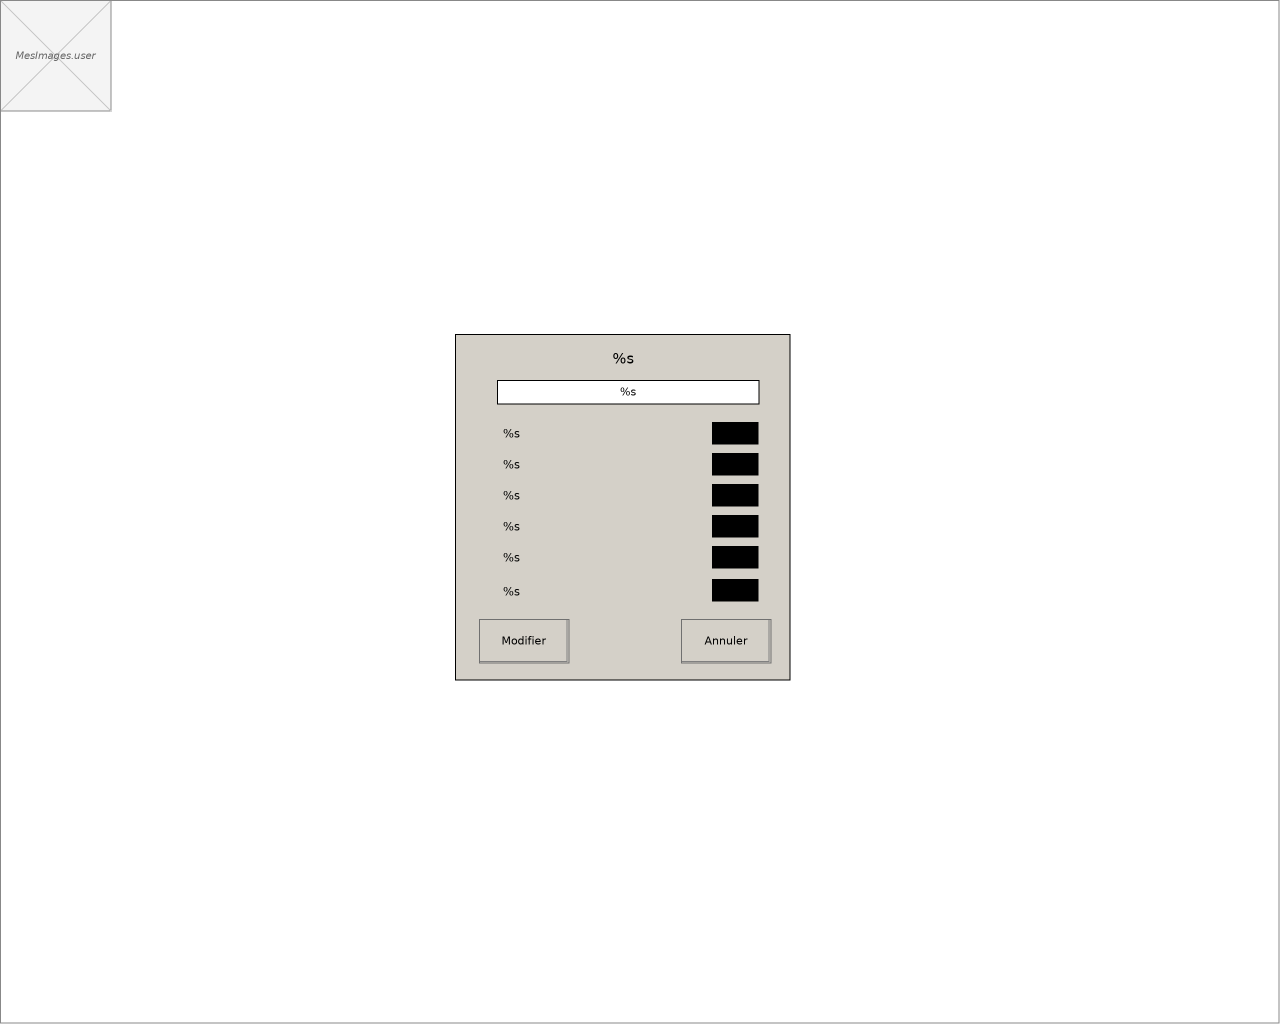
VISUALIZATION UTIL_MOD_GROUP  // 1280x1024
    Image (0,0 111x111), image: MesImages.user
    RoundedRectangle (455,334 335x346)
    Rectangle (460,344 327x29), "%s", text list: 'TextList_Util_Group', text index: 9
    Rectangle (500,450 112x29), "%s", text list: 'TextList_Util_Group', text index: 4
    Rectangle (500,481 112x29), "%s", text list: 'TextList_Util_Group', text index: 5
    Rectangle (500,419 112x29), "%s", text list: 'TextList_Util_Group', text index: 3
    Rectangle (500,512 112x29), "%s", text list: 'TextList_Util_Group', text index: 6
    Rectangle (500,543 112x29), "%s", text list: 'TextList_Util_Group', text index: 7
    Rectangle (500,577 122x29), "%s", text list: 'TextList_Util_Group', text index: 8
    Rectangle (712,422 46x22), "Oui", colour toggle: Global_Variables.PRG_USER.GROUP_TEMP.PROGRAMMATION
        toggle Global_Variables.PRG_USER.GROUP_TEMP.PROGRAMMATION
    Rectangle (712,453 46x22), "Oui", colour toggle: Global_Variables.PRG_USER.GROUP_TEMP.MAINTENANCE
        toggle Global_Variables.PRG_USER.GROUP_TEMP.MAINTENANCE
    Rectangle (712,484 46x22), "Oui", colour toggle: Global_Variables.PRG_USER.GROUP_TEMP.SUPERVISEUR
        toggle Global_Variables.PRG_USER.GROUP_TEMP.SUPERVISEUR
    Rectangle (712,515 46x22), "Oui", colour toggle: Global_Variables.PRG_USER.GROUP_TEMP.PRODUCTION
        toggle Global_Variables.PRG_USER.GROUP_TEMP.PRODUCTION
    Rectangle (712,546 46x22), "Oui", colour toggle: Global_Variables.PRG_USER.GROUP_TEMP.CONF_MACHINE
        toggle Global_Variables.PRG_USER.GROUP_TEMP.CONF_MACHINE
    Rectangle (712,579 46x22), "Oui", colour toggle: Global_Variables.PRG_USER.GROUP_TEMP.FONCTION_SA
        toggle Global_Variables.PRG_USER.GROUP_TEMP.FONCTION_SA
    Button (479,619 90x44), "Modifier", input disabled if: NOT PRG_USER.AUT_NOM_GRP
        toggle PRG_USER.DD_mod_group2
        OnMouseClick: change screen: UTIL_GROUP
    Button (681,619 90x44), "Annuler"
        OnMouseClick: change screen: UTIL_GROUP
    Rectangle (497,380 262x24), "%s", text variable: PRG_USER.GROUP_TEMP.NOM
        OnMouseClick: write the text variable via InputWithLimits
END_VISUALIZATION

// ---- Visualizations/Users/UTIL_MOD_USER.TcVIS
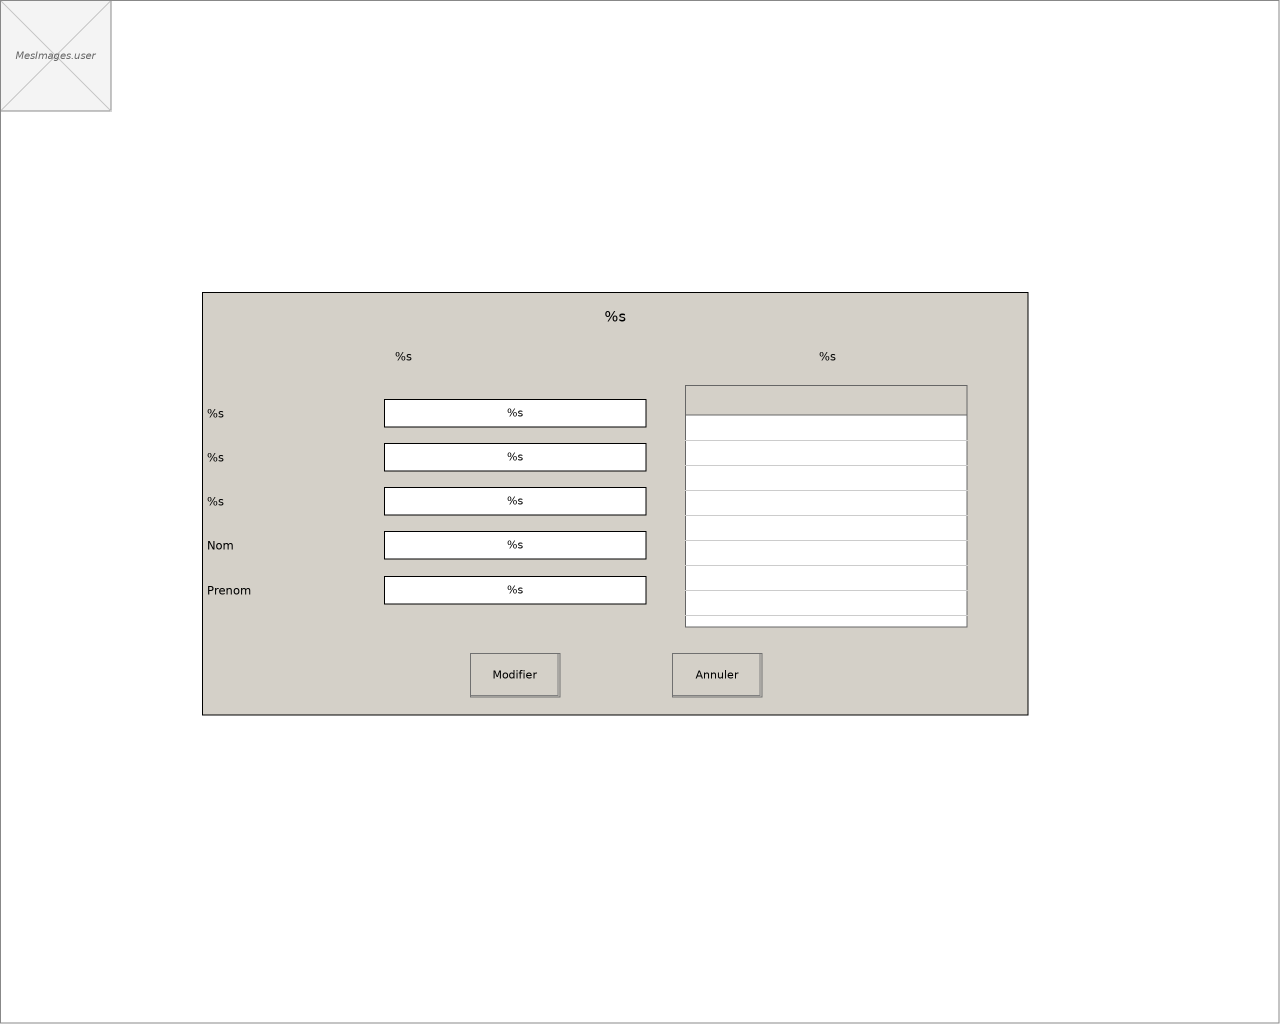
VISUALIZATION UTIL_MOD_USER  // 1280x1024
    Image (0,0 111x111), image: MesImages.user
    RoundedRectangle (202,292 826x423)
    Rectangle (206,302 819x29), "%s", text list: 'TextList_Util_Userlist', text index: 0
    Button (470,653 90x44), "Modifier", input disabled if: NOT PRG_USER.AUT_NOM_USER
        toggle PRG_USER.DD_mod_user2
        OnMouseClick: change screen: UTIL_USER
    Button (672,653 90x44), "Annuler"
        OnMouseClick: change screen: UTIL_USER
    Rectangle (384,399 262x28), "%s", text variable: PRG_USER.USER_TEMP.LOGIN
        OnMouseClick: write the text variable via InputWithLimits
    Rectangle (205,342 397x29), "%s", text list: 'TextList_Util_Userlist', text index: 2
    Rectangle (629,342 397x29), "%s", text list: 'TextList_Util_Userlist', text index: 3
    Table (685,385 282x242), data array: PRG_USER.TBL_GROUP
        p1137915858: PRG_USER.LIGNE_GROUP
        p3854506369: PRG_USER.TBL_GROUP[INDEX].NOM
        p1892666644: PRG_USER.TBL_GROUP[INDEX].PROGRAMMATION
        p338671338: PRG_USER.TBL_GROUP[INDEX].MAINTENANCE
        p2170511999: PRG_USER.TBL_GROUP[INDEX].SUPERVISEUR
        p3723444502: PRG_USER.TBL_GROUP[INDEX].PRODUCTION
        p1218418051: PRG_USER.TBL_GROUP[INDEX].CONF_MACHINE
        p746581629: PRG_USER.TBL_GROUP[INDEX].FONCTION_SA
        p3104783080: PRG_USER.TBL_GROUP[INDEX].CONF_TRF
        p2501879983: PRG_USER.TBL_GROUP[INDEX].MODIF_ENLIGNE
        p7306298: PRG_USER.TBL_GROUP[INDEX].ARCHIVE_EV
        p1933151965: PRG_USER.TBL_GROUP[INDEX].DECONSIGNATION
        p2232123230: Nom du groupe
        p511219082: Pro. Ed
        p1755163831: Maint.
        p4092479075: Superv.
        p2237128397: Prod.
        p505689113: Conf.
        p1757482276: FoncSA.
    Rectangle (204,399 173x29), "%s", text list: 'TextList_Users_Menu', text index: 5
    Rectangle (204,443 173x29), "%s", text list: 'TextList_Users_Menu', text index: 6
    Rectangle (204,487 173x29), "%s", text list: 'TextList_Users_Menu', text index: 21
    Rectangle (204,531 173x29), "Nom"
    Rectangle (204,576 173x29), "Prenom"
    Rectangle (384,443 262x28), "%s", text variable: PRG_USER.USER_TEMP.PASS
        OnMouseClick: write the text variable via InputWithLimits, password
    Rectangle (384,487 262x28), "%s", text variable: PRG_USER.PASS_CONF
        OnMouseClick: write the text variable via InputWithLimits, password
    Rectangle (384,531 262x28), "%s", text variable: PRG_USER.USER_TEMP.NOM
        OnMouseClick: write the text variable via InputWithLimits
    Rectangle (384,576 262x28), "%s", text variable: PRG_USER.USER_TEMP.PRENOM
        OnMouseClick: write the text variable via InputWithLimits
END_VISUALIZATION

// ---- Visualizations/Users/UTIL_NEW_GROUP.TcVIS
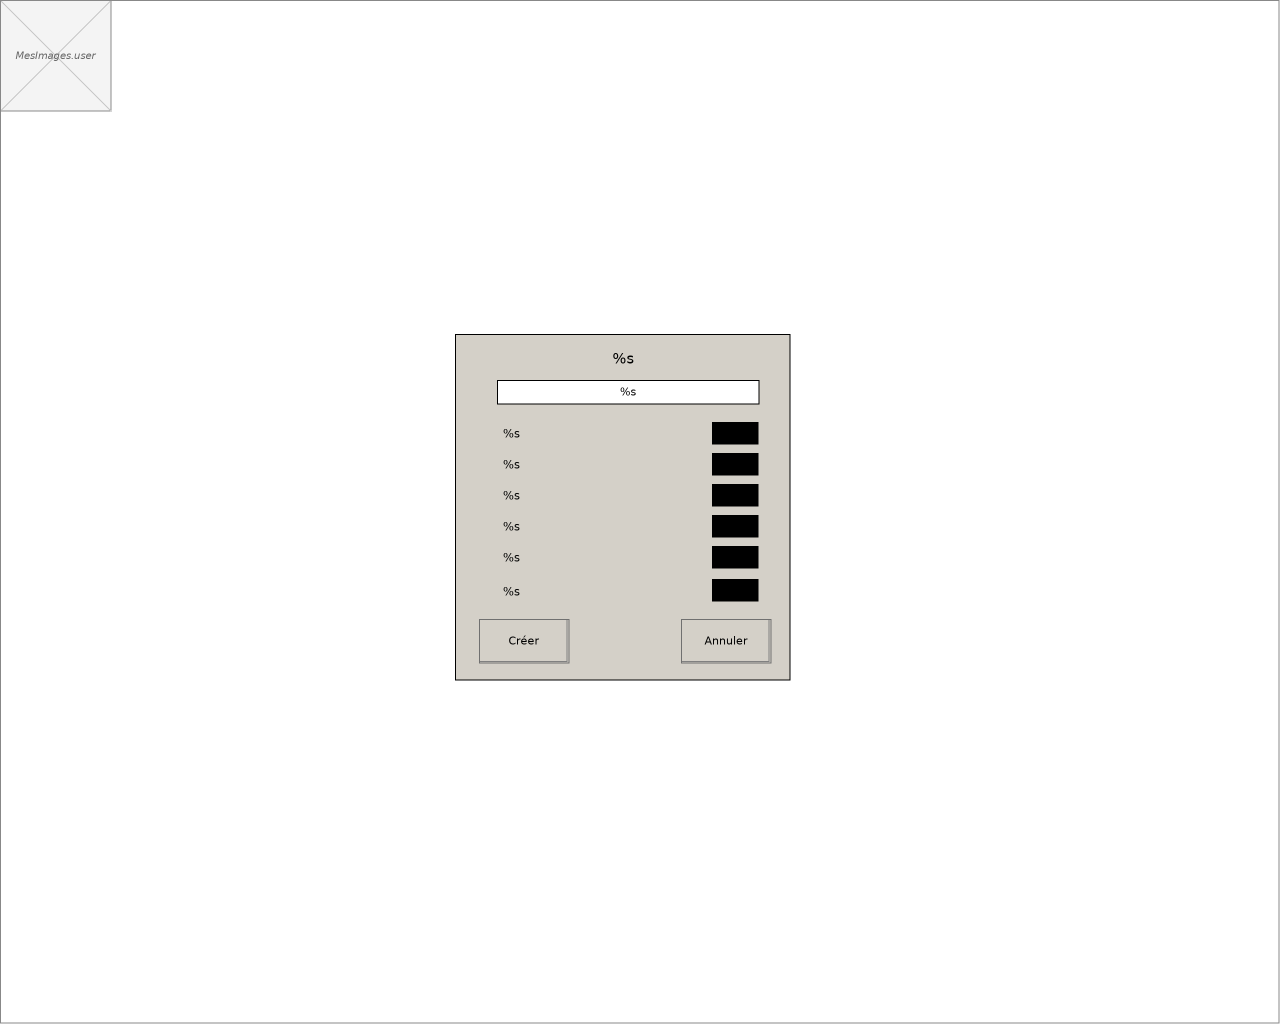
VISUALIZATION UTIL_NEW_GROUP  // 1280x1024
    Image (0,0 111x111), image: MesImages.user
    RoundedRectangle (455,334 335x346)
    Rectangle (460,344 327x29), "%s", text list: 'TextList_Util_Group', text index: 10
    Rectangle (500,450 112x29), "%s", text list: 'TextList_Util_Group', text index: 4
    Rectangle (500,481 112x29), "%s", text list: 'TextList_Util_Group', text index: 5
    Rectangle (500,419 112x29), "%s", text list: 'TextList_Util_Group', text index: 3
    Rectangle (500,512 112x29), "%s", text list: 'TextList_Util_Group', text index: 6
    Rectangle (500,543 112x29), "%s", text list: 'TextList_Util_Group', text index: 7
    Rectangle (500,577 122x29), "%s", text list: 'TextList_Util_Group', text index: 8
    Rectangle (712,422 46x22), "Oui", colour toggle: Global_Variables.PRG_USER.GROUP_TEMP.PROGRAMMATION
        toggle Global_Variables.PRG_USER.GROUP_TEMP.PROGRAMMATION
    Rectangle (712,453 46x22), "Oui", colour toggle: Global_Variables.PRG_USER.GROUP_TEMP.MAINTENANCE
        toggle Global_Variables.PRG_USER.GROUP_TEMP.MAINTENANCE
    Rectangle (712,484 46x22), "Oui", colour toggle: Global_Variables.PRG_USER.GROUP_TEMP.SUPERVISEUR
        toggle Global_Variables.PRG_USER.GROUP_TEMP.SUPERVISEUR
    Rectangle (712,515 46x22), "Oui", colour toggle: Global_Variables.PRG_USER.GROUP_TEMP.PRODUCTION
        toggle Global_Variables.PRG_USER.GROUP_TEMP.PRODUCTION
    Rectangle (712,546 46x22), "Oui", colour toggle: Global_Variables.PRG_USER.GROUP_TEMP.CONF_MACHINE
        toggle Global_Variables.PRG_USER.GROUP_TEMP.CONF_MACHINE
    Rectangle (712,579 46x22), "Oui", colour toggle: Global_Variables.PRG_USER.GROUP_TEMP.FONCTION_SA
        toggle Global_Variables.PRG_USER.GROUP_TEMP.FONCTION_SA
    Button (479,619 90x44), "Créer"
        toggle PRG_USER.DD_NEW_GROUP
        OnMouseClick: change screen: UTIL_GROUP
    Button (681,619 90x44), "Annuler"
        OnMouseClick: change screen: UTIL_GROUP
    Rectangle (497,380 262x24), "%s", text variable: PRG_USER.GROUP_TEMP.NOM
        OnMouseClick: write the text variable via InputWithLimits
END_VISUALIZATION

// ---- Visualizations/Users/UTIL_NEW_USER.TcVIS
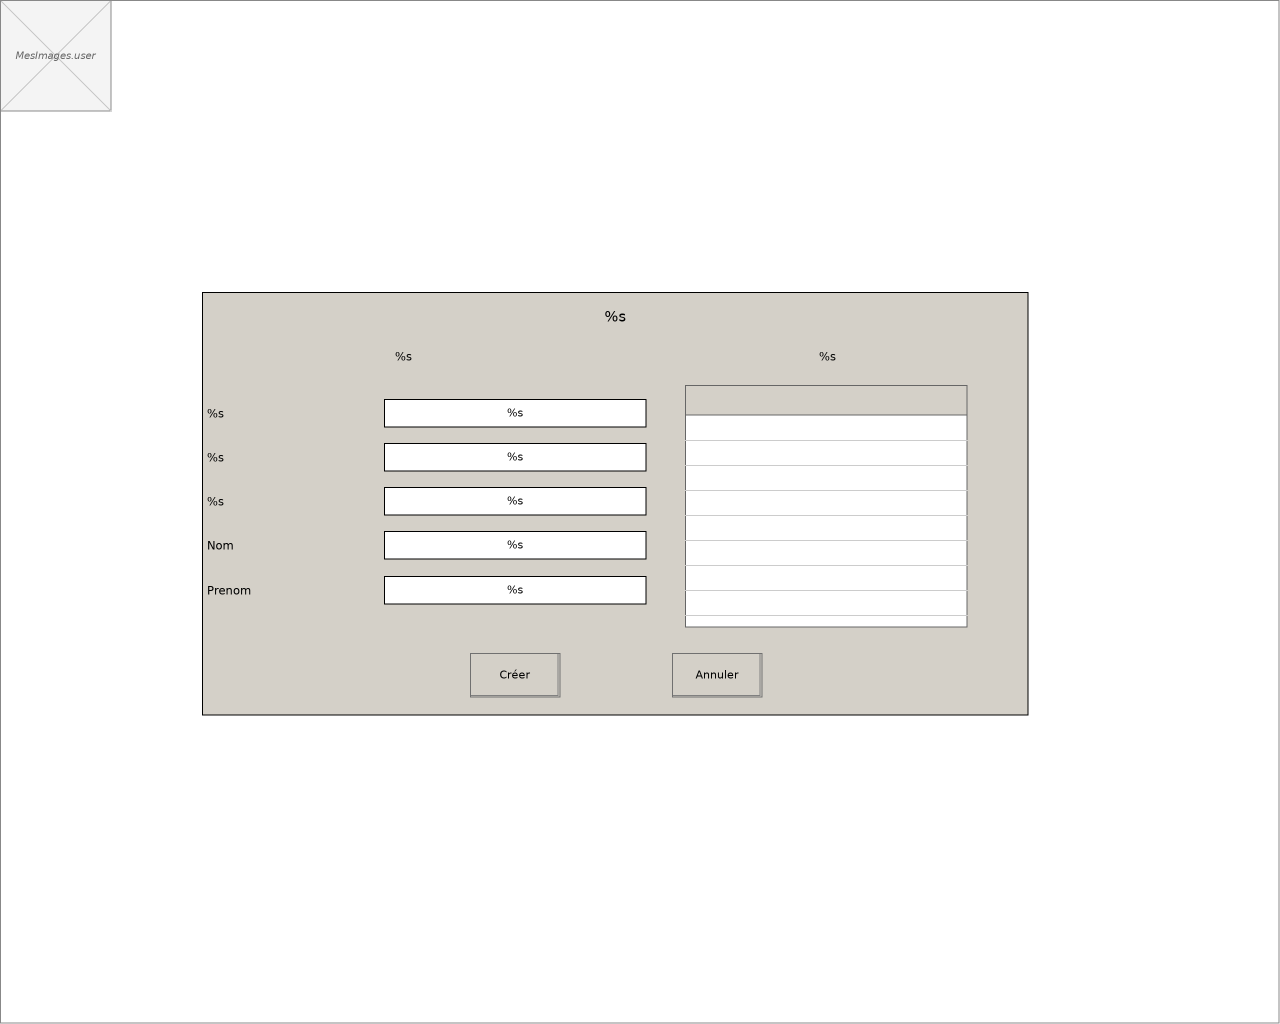
VISUALIZATION UTIL_NEW_USER  // 1280x1024
    Image (0,0 111x111), image: MesImages.user
    RoundedRectangle (202,292 826x423)
    Rectangle (206,302 819x29), "%s", text list: 'TextList_Util_Userlist', text index: 1
    Button (470,653 90x44), "Créer", input disabled if: NOT PRG_USER.AUT_NEW_USER
        toggle PRG_USER.DD_NEW_USER
        OnMouseClick: change screen: UTIL_USER
    Button (672,653 90x44), "Annuler"
        OnMouseClick: change screen: UTIL_USER
    Rectangle (384,399 262x28), "%s", text variable: PRG_USER.USER_TEMP.LOGIN
        OnMouseClick: write the text variable via InputWithLimits
    Rectangle (205,342 397x29), "%s", text list: 'TextList_Util_Userlist', text index: 2
    Rectangle (629,342 397x29), "%s", text list: 'TextList_Util_Userlist', text index: 3
    Table (685,385 282x242), data array: PRG_USER.TBL_GROUP
        p1137915858: PRG_USER.LIGNE_GROUP
        p3854506369: PRG_USER.TBL_GROUP[INDEX].NOM
        p1892666644: PRG_USER.TBL_GROUP[INDEX].PROGRAMMATION
        p338671338: PRG_USER.TBL_GROUP[INDEX].MAINTENANCE
        p2170511999: PRG_USER.TBL_GROUP[INDEX].SUPERVISEUR
        p3723444502: PRG_USER.TBL_GROUP[INDEX].PRODUCTION
        p1218418051: PRG_USER.TBL_GROUP[INDEX].CONF_MACHINE
        p746581629: PRG_USER.TBL_GROUP[INDEX].FONCTION_SA
        p3104783080: PRG_USER.TBL_GROUP[INDEX].CONF_TRF
        p2501879983: PRG_USER.TBL_GROUP[INDEX].MODIF_ENLIGNE
        p7306298: PRG_USER.TBL_GROUP[INDEX].ARCHIVE_EV
        p1933151965: PRG_USER.TBL_GROUP[INDEX].DECONSIGNATION
        p2232123230: Nom du groupe
        p511219082: Pro. Ed
        p1755163831: Maint.
        p4092479075: Superv.
        p2237128397: Prod.
        p505689113: Conf.
        p1757482276: FoncSA.
    Rectangle (204,399 173x29), "%s", text list: 'TextList_Users_Menu', text index: 5
    Rectangle (204,443 173x29), "%s", text list: 'TextList_Users_Menu', text index: 6
    Rectangle (204,487 173x29), "%s", text list: 'TextList_Users_Menu', text index: 21
    Rectangle (204,531 173x29), "Nom"
    Rectangle (204,576 173x29), "Prenom"
    Rectangle (384,443 262x28), "%s", text variable: PRG_USER.USER_TEMP.PASS_DISPLAY
        OnMouseClick: write PRG_USER.USER_TEMP.PASS via InputWithLimits, password
    Rectangle (384,487 262x28), "%s", text variable: PRG_USER.PASS_CONF_DISPLAY
        OnMouseClick: write PRG_USER.PASS_CONF via InputWithLimits, password
    Rectangle (384,531 262x28), "%s", text variable: PRG_USER.USER_TEMP.NOM
        OnMouseClick: write the text variable via InputWithLimits
    Rectangle (384,576 262x28), "%s", text variable: PRG_USER.USER_TEMP.PRENOM
        OnMouseClick: write the text variable via InputWithLimits
END_VISUALIZATION

// ---- Visualizations/Users/UTIL_OPT.TcVIS
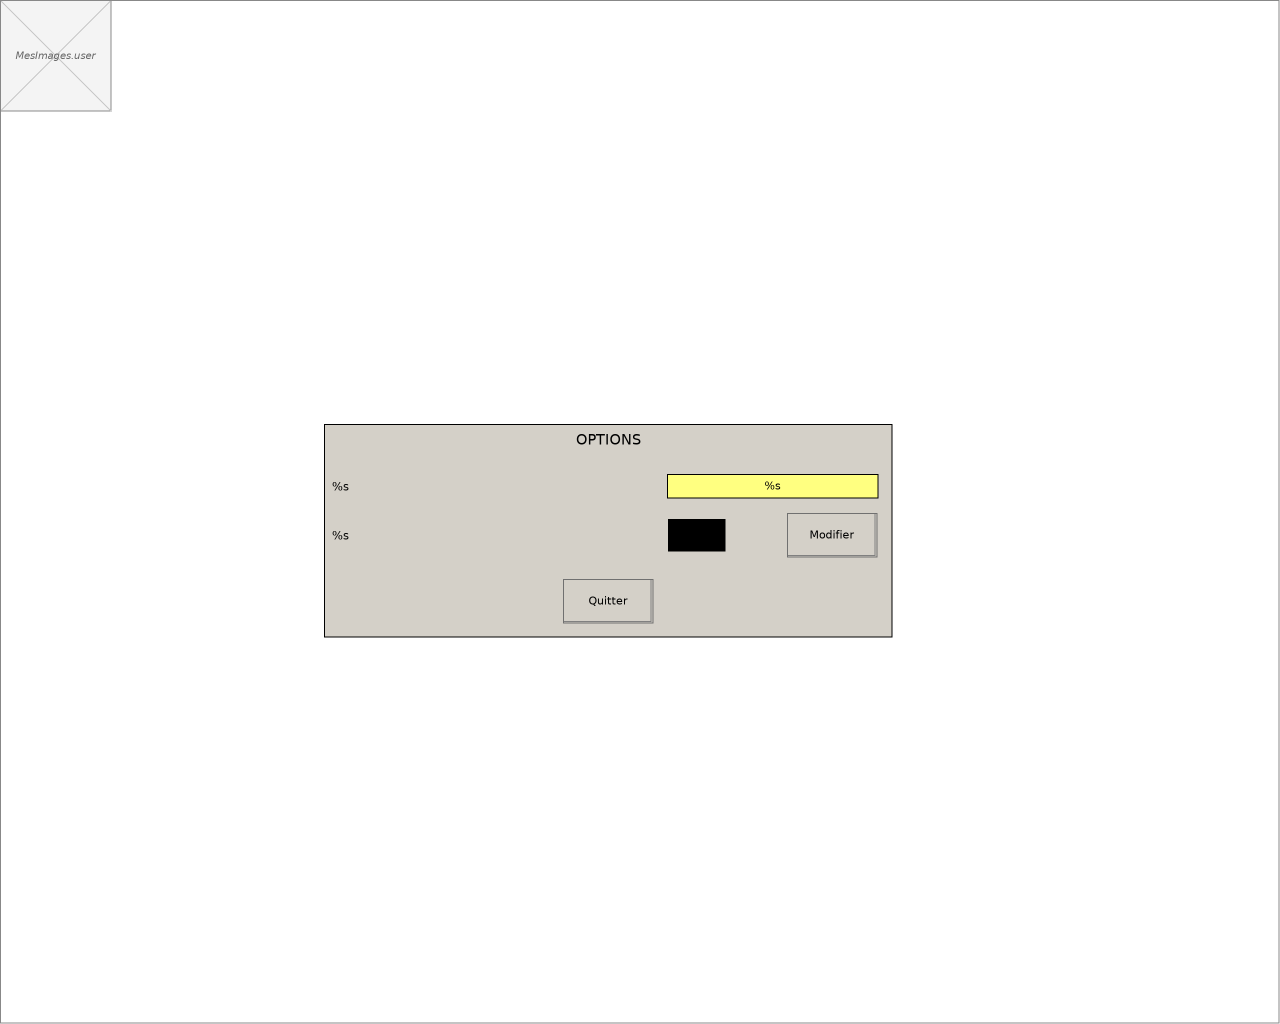
VISUALIZATION UTIL_OPT  // 1280x1024
    Image (0,0 111x111), image: MesImages.user
    RoundedRectangle (324,424 568x213)
    Rectangle (346,425 525x29), "OPTIONS"
    Button (563,579 90x44), "Quitter"
        toggle RQ_PARAM_SYSTEM
        OnMouseClick: change screen: UTIL_MENU
    Rectangle (329,472 295x29), "%s", text list: 'TextList_Users_Menu', text index: 30
    Rectangle (667,474 211x24), "%s", text variable: PRG_USER.TIM_LOGOUT
        OnMouseClick: write the text variable via InputWithLimits
    Rectangle (329,521 295x29), "%s", text list: 'TextList_Users_Menu', text index: 31
    Rectangle (668,519 57x32), "Oui", colour toggle: PRG_USER.OPT_LOGOUT
    Button (787,513 90x44), "Modifier"
        toggle PRG_USER.OPT_LOGOUT
END_VISUALIZATION

// ---- Visualizations/Users/UTIL_USER.TcVIS
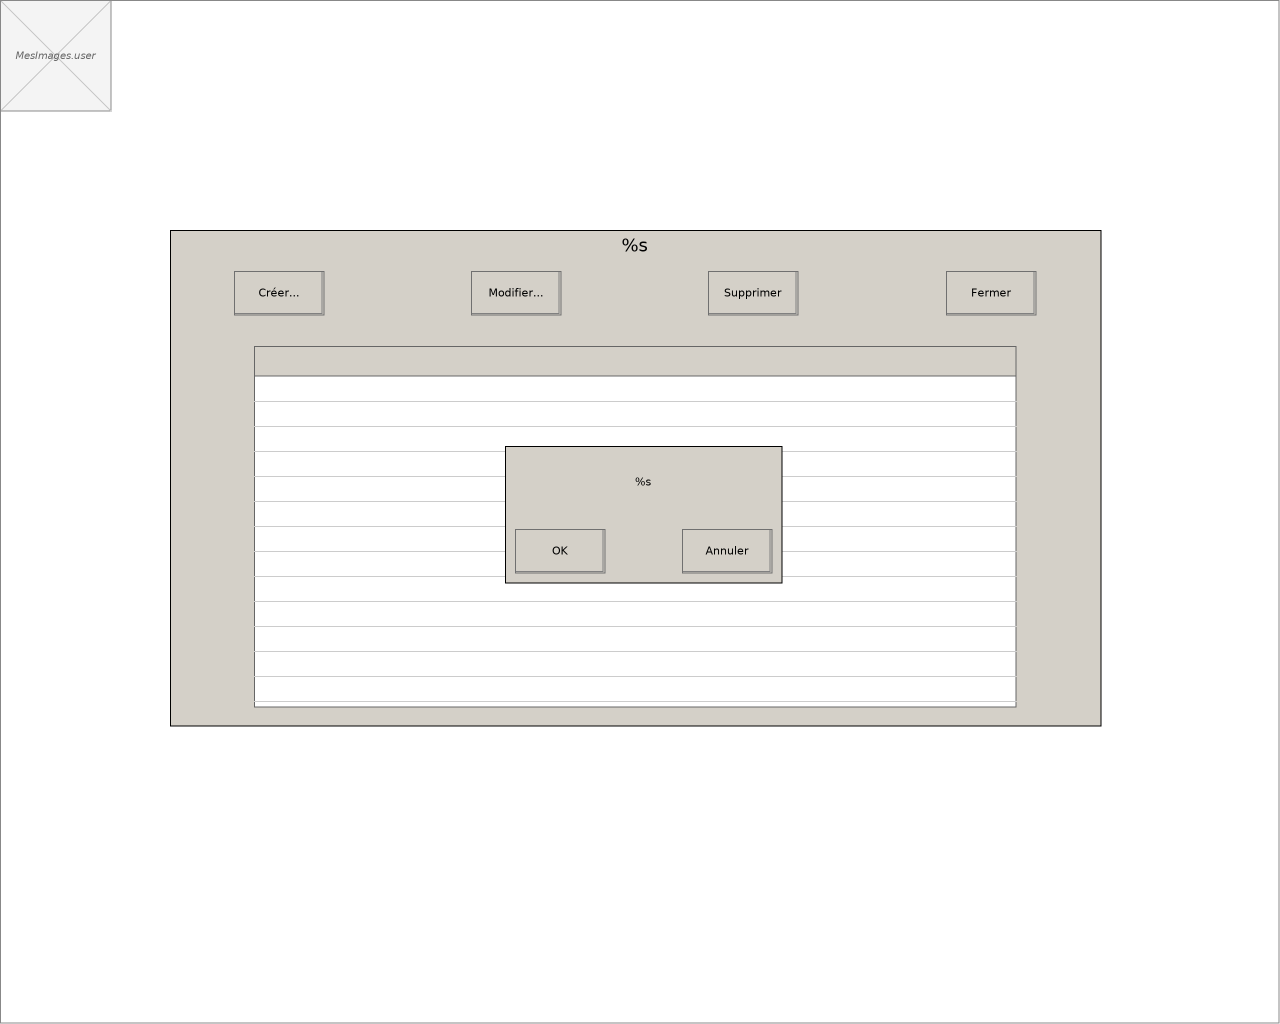
VISUALIZATION UTIL_USER  // 1280x1024
    RoundedRectangle (170,230 931x496)
    Image (0,0 111x111), image: MesImages.user
    Table (254,346 762x361), data array: PRG_USER.TBL_USER
        p1137915858: PRG_USER.LIGNE
        p3854506369: PRG_USER.TBL_USER[INDEX].LOGIN
        p1892666644: PRG_USER.TBL_USER[INDEX].PASS
        p338671338: PRG_USER.TBL_USER[INDEX].PASS_DISPLAY
        p2170511999: PRG_USER.TBL_USER[INDEX].NOM
        p3723444502: PRG_USER.TBL_USER[INDEX].PRENOM
        p1218418051: PRG_USER.TBL_USER[INDEX].GROUPE
        p2232123230: Identifiant
        p4092479075: Nom
        p2237128397: Prenom
        p505689113: Groupe
    Textfield (231,233 808x25), "%s", text list: 'TextList_Util_Userlist', text index: 4
    Button (234,271 90x44), "Créer...", invisible if: PRG_USER.STOP_USER
        toggle PRG_USER.DD_EFFACE_NEW
        OnMouseClick: change screen: UTIL_NEW_USER
    Button (471,271 90x44), "Modifier...", input disabled if: NOT PRG_USER.AUT_MOD_USER
        toggle PRG_USER.DD_mod_user1
        OnMouseClick: change screen: UTIL_MOD_USER
    Button (708,271 90x44), "Supprimer", input disabled if: NOT PRG_USER.AUT_MOD_USER
        toggle PRG_USER.VISU_FEN3
    Button (946,271 90x44), "Fermer", input disabled if: PRG_USER.VISU_FEN3
        OnMouseClick: change screen: UTIL_MENU
    Frame (505,446 280x139), invisible if: NOT PRG_USER.VISU_FEN3
        shows UTIL_CONFIRM(Num_Text := 18, OrdreDD := PRG_USER.DD_DEL_USER, Visu := PRG_USER.VISU_FEN3)
END_VISUALIZATION
